PROGRAM POU_writeSeparatorToSupvData
VAR
	sNetId: T_AmsNetId := SUPVams.sNetId;	// '5.30.23.91.1.1';
	nPort: T_AmsPort := SUPVams.nPort; 		// 851	

	FB_WriteAmsValue_XMEAS: FB_WriteAmsValue;
	FB_WriteAmsValue_XMV: FB_WriteAmsValue;
	nXMEASWriteErrorId: UDINT;
	bXMEASWriteError: BOOL;
	bXMVWriteError: BOOL;
	nXMVWriteErrorId: UDINT;
END_VAR

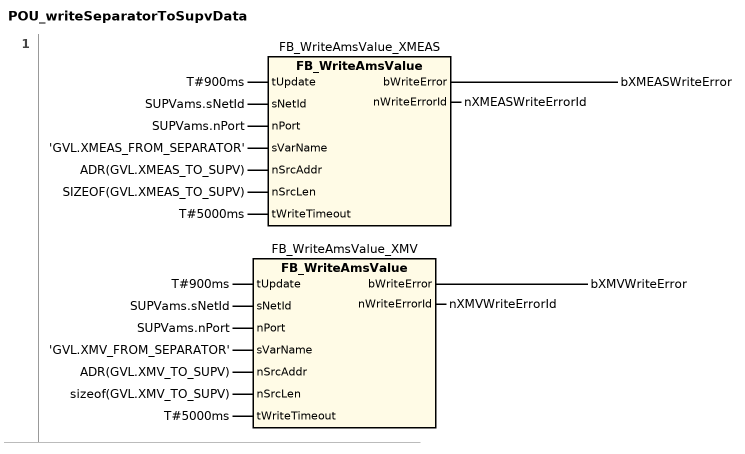
// NETWORK 1
FB_WriteAmsValue_XMEAS(
    tUpdate := T#900ms,
    sNetId := SUPVams.sNetId,
    nPort := SUPVams.nPort,
    sVarName := 'GVL.XMEAS_FROM_SEPARATOR',
    nSrcAddr := ADR(GVL.XMEAS_TO_SUPV),
    nSrcLen := SIZEOF(GVL.XMEAS_TO_SUPV),
    tWriteTimeout := T#5000ms,
    nWriteErrorId => nXMEASWriteErrorId); // FB_WriteAmsValue
bXMEASWriteError := FB_WriteAmsValue_XMEAS.bWriteError;
FB_WriteAmsValue_XMV(
    tUpdate := T#900ms,
    sNetId := SUPVams.sNetId,
    nPort := SUPVams.nPort,
    sVarName := 'GVL.XMV_FROM_SEPARATOR',
    nSrcAddr := ADR(GVL.XMV_TO_SUPV),
    nSrcLen := sizeof(GVL.XMV_TO_SUPV),
    tWriteTimeout := T#5000ms,
    nWriteErrorId => nXMVWriteErrorId); // FB_WriteAmsValue
bXMVWriteError := FB_WriteAmsValue_XMV.bWriteError;

END_PROGRAM

(* stored: Version 1.1.0.1, ProductVersion 3.1.4024.11
   POU POU_writeSeparatorToSupvData: Id {5e7ac2b2-7ed4-47ff-8a64-ec6be7ac94e9}, SpecialFunc None *)
